(* IEC 61131-3 sources: lasal-git-demo/CPU/LasalDemoProject/Class/TO161, 1 file *)

(* ---- TO161.st ---- *)
#define DEVICE_ID_TO161 1004

#define TO161_ADDR_CYC_WRITE  0
#define TO161_ADDR_CYC_READ   2

#define TO161_WRITE_LENGTH    2
#define TO161_READ_LENGTH     2

(*!
<Class
	Name               = "TO161"
	Revision           = "1.34"
	RealtimeTask       = "false"
	CyclicTask         = "false"
	BackgroundTask     = "false"
	Sigmatek           = "true"
	OSInterface        = "false"
	HighPriority       = "false"
	Automatic          = "false"
	UpdateMode         = "Prescan"
	IconPath           = ".\Class\s-dias.ico"
	SharedCommandTable = "true"
	Objectsize         = "(494,120)"
	Comment            = "This hardware class is used to control the TO161 hardware module with 16 digital outputs.">
	<Channels>
		<Server Name="Output1" Visualized="true" Initialize="false" WriteProtected="false" Retentive="false" Comment="Digital Output 1"/>
		<Server Name="Output10" Visualized="true" Initialize="false" WriteProtected="false" Retentive="false" Comment="Digital Output 10"/>
		<Server Name="Output11" Visualized="true" Initialize="false" WriteProtected="false" Retentive="false" Comment="Digital Output 11"/>
		<Server Name="Output12" Visualized="true" Initialize="false" WriteProtected="false" Retentive="false" Comment="Digital Output 12"/>
		<Server Name="Output13" Visualized="true" Initialize="false" WriteProtected="false" Retentive="false" Comment="Digital Output 13"/>
		<Server Name="Output14" Visualized="true" Initialize="false" WriteProtected="false" Retentive="false" Comment="Digital Output 14"/>
		<Server Name="Output15" Visualized="true" Initialize="false" WriteProtected="false" Retentive="false" Comment="Digital Output 15"/>
		<Server Name="Output16" Visualized="true" Initialize="false" WriteProtected="false" Retentive="false" Comment="Digital Output 16"/>
		<Server Name="Output2" Visualized="true" Initialize="false" WriteProtected="false" Retentive="false" Comment="Digital Output 2"/>
		<Server Name="Output3" Visualized="true" Initialize="false" WriteProtected="false" Retentive="false" Comment="Digital Output 3"/>
		<Server Name="Output4" Visualized="true" Initialize="false" WriteProtected="false" Retentive="false" Comment="Digital Output 4"/>
		<Server Name="Output5" Visualized="true" Initialize="false" WriteProtected="false" Retentive="false" Comment="Digital Output 5"/>
		<Server Name="Output6" Visualized="true" Initialize="false" WriteProtected="false" Retentive="false" Comment="Digital Output 6"/>
		<Server Name="Output7" Visualized="true" Initialize="false" WriteProtected="false" Retentive="false" Comment="Digital Output 7"/>
		<Server Name="Output8" Visualized="true" Initialize="false" WriteProtected="false" Retentive="false" Comment="Digital Output 8"/>
		<Server Name="Output9" Visualized="true" Initialize="false" WriteProtected="false" Retentive="false" Comment="Digital Output 9"/>
		<Server Name="OutputWord" Visualized="true" Initialize="false" WriteProtected="false" Retentive="false" Comment="The digital outputs are displayed in this server in a 16-bit field"/>
		<Server Name="VoltageOkBank1" Visualized="true" Initialize="false" WriteProtected="true" Retentive="false" Comment="Supply voltage ok&#13;&#10;+24V1 (Digital Out 1-8)"/>
		<Server Name="VoltageOkBank2" Visualized="true" Initialize="false" WriteProtected="true" Retentive="false" Comment="Supply voltage ok&#13;&#10;+24V2 (Digital Out 9-16)"/>
	</Channels>
	<RevDoku>
		<Owner Company="Sigmatek" Author="BeiWol"/>
		<Dokumentation Revision="1.34" Date="12.08.2019" Author="LazJos" Company="Sigmatek" Description="Added support for HWAlarms."/>
		<Dokumentation Revision="1.33" Date="09.01.2019" Author="FurDom" Company="Sigmatek" Description="Added function for Spi Write in SdiasBase class."/>
		<Dokumentation Revision="1.32" Date="08.06.2018" Author="RamAnd" Company="Sigmatek" Description="LASAL Hardware Description (.lhd) file has been updated."/>
		<Dokumentation Revision="1.31" Date="16.05.2017" Author="RamAnd" Company="Sigmatek" Description="When adding an SDO (i.e. via ReadSPIData) from background priority it was possible that the adding process got interrupted by receiving the answer to this SDO which is handled in cyclic priority. In the error case the answer was unexpected and therefore ignored. Then the class signals a timeout while waiting for the answer, which already arrived before waiting for it. Added mutex and changed instruction order to prevent this error."/>
		<Dokumentation Revision="1.30" Date="12.07.2016" Author="SeiChr" Company="Sigmatek" Description="Added Values for the total Current calculation. SA 31571"/>
		<Dokumentation Revision="1.29" Date="01.03.2016" Author="EisMic" Company="Sigmatek" Description="Corrected BoundExceed Error in base class at Write method of LEDControl Server when Place = LSL_DEACTIVATED."/>
		<Dokumentation Revision="1.28" Date="22.06.2015" Author="EisMic" Company="Sigmatek" Description="The servers FPGAVersion, SerialNo, Device ID and status and input servers are now not reset anymore when the module is disconnected.&#13;&#10;Outputs are now written to the hardware in any case after a reconnect."/>
		<Dokumentation Revision="1.27" Date="27.05.2015" Author="EisMic" Company="Sigmatek" Description="Corrected ConnectEvent Method that outputs are set after reconnect."/>
		<Dokumentation Revision="1.26" Date="16.04.2015" Author="EisMic&#13;&#10;LanSte" Company="Sigmatek" Description="Added support for visualisation in graphical hardware editor.&#13;&#10;Added support for calculating resources for graphical hardware editor."/>
		<Dokumentation Revision="1.25" Date="17.03.2015" Author="RamAnd" Company="Sigmatek" Description="Added HW Version for sdias clients."/>
		<Dokumentation Revision="1.24" Date="11.02.2015" Author="PieSte" Company="Sigmatek" Description="Corrected read spi data for hardwaretree in methode GetSPIDataFromID from baseclass."/>
		<Dokumentation Revision="1.23" Date="03.12.2014" Author="PieSte" Company="Sigmatek" Description="Add OutputByte in .lhd file."/>
		<Dokumentation Revision="1.22" Date="18.11.2014" Author="PieSte" Company="Sigmatek" Description="Added possibility  to read more data from spi flash then one sdo access.&#13;&#10;Set methode GetDeviceID to global.&#13;&#10;Add methode to calculate checksum of spi flash."/>
		<Dokumentation Revision="1.21" Date="09.07.2014" Author="EisMic" Company="Sigmatek" Description="Added support for reading hardware diagnosis and hardwaretree entry."/>
		<Dokumentation Revision="1.20" Date="20.01.2014" Author="PieSte" Company="Sigmatek" Description="Read Client Required and Place in Init SdiasBase"/>
		<Dokumentation Revision="1.10" Date="05.12.2013" Author="RamAnd" Company="Sigmatek" Description="Changed login mechanism to sdias manager class to be independent of bus accesses."/>
		<Dokumentation Revision="1.0" Date="25.07.2013" Author="BeiWol" Company="Sigmatek" Description="First library version"/>
	</RevDoku>
	<Network Name="TO161">
		<!-- List of Components in this network -->
		<Components>
			<Object
				Name       = "_base"
				Class      = "SdiasBase"
				Position   = "(218,120)"
				Visualized = "true">
				<Channels>
					<Server Name="ClassState"/>
					<Server Name="DeviceID"/>
					<Server Name="FPGAVersion"/>
					<Server Name="HwVersion"/>
					<Server Name="LEDControl" Value="0"/>
					<Server Name="RetryCounter"/>
					<Server Name="SDOState"/>
					<Server Name="SerialNo"/>
					<Client Name="Place" Value="0"/>
					<Client Name="Required" Value="1"/>
					<Client Name="SdiasIn"/>
					<Client Name="ToStdLib"/>
				</Channels>
			</Object>
		</Components>
		<Comments>
		</Comments>
		<!-- List of Connections in this network -->
		<Connections>
			<Connection Source="this.ClassState" Destination="_base.ClassState" Vertices="(804,210),(632,210),"/>
			<Connection Source="this.DeviceID" Destination="_base.DeviceID" Vertices="(804,270),(632,270),"/>
			<Connection Source="this.SerialNo" Destination="_base.SerialNo" Vertices="(804,450),(632,450),"/>
			<Connection Source="this.RetryCounter" Destination="_base.RetryCounter" Vertices="(804,510),(632,510),"/>
			<Connection Source="_base.SdiasIn" Destination="this.SdiasIn" Vertices="(218,210),(38,210),"/>
			<Connection Source="_base.Place" Destination="this.Place" Vertices="(218,270),(38,270),"/>
			<Connection Source="_base.Required" Destination="this.Required" Vertices="(218,330),(38,330),"/>
			<Connection Source="this.LEDControl" Destination="_base.LEDControl" Vertices="(804,570),(632,570),"/>
			<Connection Source="this.FPGAVersion" Destination="_base.FPGAVersion" Vertices="(804,330),(632,330),"/>
			<Connection Source="this.HwVersion" Destination="_base.HwVersion" Vertices="(804,390),(632,390),"/>
		</Connections>
		<!-- Headerfiles -->
		<Options>
		</Options>
	</Network>
</Class>
*)
#pragma using SdiasBase

TO161 : CLASS
: SdiasBase
	TYPE
	  t_VoltageOk : BINT
	  [
	    1 Ok24V1,
	    2 Ok24V2,
	  ];
	END_TYPE
  //Servers:
	Output1 	: SvrCh_DINT;
	Output2 	: SvrCh_DINT;
	Output3 	: SvrCh_DINT;
	Output4 	: SvrCh_DINT;
	Output5 	: SvrCh_DINT;
	Output6 	: SvrCh_DINT;
	Output7 	: SvrCh_DINT;
	Output8 	: SvrCh_DINT;
	Output9 	: SvrCh_DINT;
	Output10 	: SvrCh_DINT;
	Output11 	: SvrCh_DINT;
	Output12 	: SvrCh_DINT;
	Output13 	: SvrCh_DINT;
	Output14 	: SvrCh_DINT;
	Output15 	: SvrCh_DINT;
	Output16 	: SvrCh_DINT;
	OutputWord 	: SvrCh_BDINT;
	VoltageOkBank1 	: SvrCh_DINT;
	VoltageOkBank2 	: SvrCh_DINT;
  //Clients:
  //Variables:
		bdOutputBitsOld : BDINT
		[
		];
			//! <Variable Comment="Merker for old OutputStatus." Name="bdOutputBitsOld"/>
		pReadData 	: ^UINT;			//! <Variable Comment="Read-Data from the Module." Name="pReadData"/>
		pWriteData 	: ^UINT;			//! <Variable Comment="WriteData of the Module." Name="pWriteData"/>
  //Functions:
				//! <Function Comment="Realtime Update Methode which runs in PreScan." Name="UpdateRt"/>
	FUNCTION VIRTUAL GLOBAL UpdateRt;
				//! <Function Comment="Realtime Update Methode which runs in PostScan." Name="UpdateRtPostScan"/>
	FUNCTION VIRTUAL GLOBAL UpdateRtPostScan;
				//! <Function Comment="Methode is called if this Module gets connected." Name="ConnectEvent"/>
	FUNCTION VIRTUAL GLOBAL ConnectEvent;
				//! <Function Comment="Methode is called if this Module gets disconnected." Name="DisconnectEvent"/>
	FUNCTION VIRTUAL GLOBAL DisconnectEvent;
				//! <Function Comment="This Methode should is used, to check the DeviceID of the Module." Name="CheckDeviceID"/>
	FUNCTION VIRTUAL GLOBAL CheckDeviceID
		VAR_INPUT
			udID2Check 	: UDINT;			//! <Variable Comment="Device ID of connected Module." Name="CheckDeviceID.udID2Check"/>
		END_VAR
		VAR_OUTPUT
			bIsOK 	: BOOL;			//! <Variable Comment="FALSE = Wrong DeviceID for Module&#13;&#10;TRUE  = DeviceID of Module is correct" Name="CheckDeviceID.bIsOK"/>
		END_VAR;

	FUNCTION VIRTUAL GetTaskCfg
		VAR_OUTPUT
			TaskCfg 	: BDINT;			//! <Variable Comment="Select which tasks will be available for this module:&#13;&#10;Bit0..Realtime PreScan&#13;&#10;Bit1..Realtime PostScan&#13;&#10;Bit2..Cyclic&#13;&#10;&#13;&#10;e.g. if only realtime postscan is needed:&#13;&#10;2#010" Name="GetTaskCfg.TaskCfg"/>
		END_VAR;

	FUNCTION VIRTUAL GetDeviceID
		VAR_OUTPUT
			output 	: UDINT;
		END_VAR;

	FUNCTION VIRTUAL GLOBAL Output1::Write
		VAR_INPUT
			input (EAX) 	: DINT;
		END_VAR
		VAR_OUTPUT
			result (EAX) 	: DINT;
		END_VAR;

	FUNCTION VIRTUAL GLOBAL Output2::Write
		VAR_INPUT
			input (EAX) 	: DINT;
		END_VAR
		VAR_OUTPUT
			result (EAX) 	: DINT;
		END_VAR;

	FUNCTION VIRTUAL GLOBAL Output3::Write
		VAR_INPUT
			input (EAX) 	: DINT;
		END_VAR
		VAR_OUTPUT
			result (EAX) 	: DINT;
		END_VAR;

	FUNCTION VIRTUAL GLOBAL Output4::Write
		VAR_INPUT
			input (EAX) 	: DINT;
		END_VAR
		VAR_OUTPUT
			result (EAX) 	: DINT;
		END_VAR;

	FUNCTION VIRTUAL GLOBAL Output5::Write
		VAR_INPUT
			input (EAX) 	: DINT;
		END_VAR
		VAR_OUTPUT
			result (EAX) 	: DINT;
		END_VAR;

	FUNCTION VIRTUAL GLOBAL Output6::Write
		VAR_INPUT
			input (EAX) 	: DINT;
		END_VAR
		VAR_OUTPUT
			result (EAX) 	: DINT;
		END_VAR;

	FUNCTION VIRTUAL GLOBAL Output7::Write
		VAR_INPUT
			input (EAX) 	: DINT;
		END_VAR
		VAR_OUTPUT
			result (EAX) 	: DINT;
		END_VAR;

	FUNCTION VIRTUAL GLOBAL Output8::Write
		VAR_INPUT
			input (EAX) 	: DINT;
		END_VAR
		VAR_OUTPUT
			result (EAX) 	: DINT;
		END_VAR;

	FUNCTION VIRTUAL GLOBAL Output9::Write
		VAR_INPUT
			input (EAX) 	: DINT;
		END_VAR
		VAR_OUTPUT
			result (EAX) 	: DINT;
		END_VAR;

	FUNCTION VIRTUAL GLOBAL Output10::Write
		VAR_INPUT
			input (EAX) 	: DINT;
		END_VAR
		VAR_OUTPUT
			result (EAX) 	: DINT;
		END_VAR;

	FUNCTION VIRTUAL GLOBAL Output11::Write
		VAR_INPUT
			input (EAX) 	: DINT;
		END_VAR
		VAR_OUTPUT
			result (EAX) 	: DINT;
		END_VAR;

	FUNCTION VIRTUAL GLOBAL Output12::Write
		VAR_INPUT
			input (EAX) 	: DINT;
		END_VAR
		VAR_OUTPUT
			result (EAX) 	: DINT;
		END_VAR;

	FUNCTION VIRTUAL GLOBAL Output13::Write
		VAR_INPUT
			input (EAX) 	: DINT;
		END_VAR
		VAR_OUTPUT
			result (EAX) 	: DINT;
		END_VAR;

	FUNCTION VIRTUAL GLOBAL Output14::Write
		VAR_INPUT
			input (EAX) 	: DINT;
		END_VAR
		VAR_OUTPUT
			result (EAX) 	: DINT;
		END_VAR;

	FUNCTION VIRTUAL GLOBAL Output15::Write
		VAR_INPUT
			input (EAX) 	: DINT;
		END_VAR
		VAR_OUTPUT
			result (EAX) 	: DINT;
		END_VAR;

	FUNCTION VIRTUAL GLOBAL Output16::Write
		VAR_INPUT
			input (EAX) 	: DINT;
		END_VAR
		VAR_OUTPUT
			result (EAX) 	: DINT;
		END_VAR;

	FUNCTION VIRTUAL GLOBAL OutputWord::Write
		VAR_INPUT
			input (EAX) 	: BDINT;
		END_VAR
		VAR_OUTPUT
			result (EAX) 	: BDINT;
		END_VAR;
  //Tables:
	FUNCTION @STD
		VAR_OUTPUT
			ret_code	: CONFSTATES;
		END_VAR;
	FUNCTION GLOBAL TAB @CT_;
END_CLASS;

FUNCTION VIRTUAL GLOBAL TO161::UpdateRt
  VAR
    VoltageOkTmp  : t_VoltageOk;
  END_VAR

  VoltageOkTmp := (pReadData^)$BINT;

  VoltageOkBank1 := VoltageOkTmp.Ok24V1;
  VoltageOkBank2 := VoltageOkTmp.Ok24V2;

END_FUNCTION

FUNCTION VIRTUAL GLOBAL TO161::UpdateRtPostScan

  if OutputWord <> bdOutputBitsOld then
    pWriteData^ := OutputWord$BINT;

    bdOutputBitsOld := OutputWord;
  end_if;

END_FUNCTION

FUNCTION VIRTUAL GLOBAL TO161::CheckDeviceID
	VAR_INPUT
		udID2Check 	: UDINT;
	END_VAR
	VAR_OUTPUT
		bIsOK 	: BOOL;
	END_VAR

  //look if it is right hardware
	if ( udID2Check <> DEVICE_ID_TO161 ) then
		bIsOK := FALSE;
	else
    bIsOK := TRUE;
	end_if;

END_FUNCTION

FUNCTION VIRTUAL GLOBAL TO161::ConnectEvent

  // start the accesses on the SDIAS (initialize the control byte in the DPRAM)
  if DefaultAccesses.ReadAccess.pControlByte then
    pReadData := DefaultAccesses.ReadAccess.pData$^UINT;

    DefaultAccesses.ReadAccess.pControlByte^.EnableDO := TRUE;
  else
    eInitState := _DOHandleInvalid;
    return;
  end_if;

  if DefaultAccesses.WriteAccess.pControlByte then
    pWriteData := DefaultAccesses.WriteAccess.pData$^UINT;

    DefaultAccesses.WriteAccess.pControlByte^.EnableDO := TRUE;
  else
    eInitState := _DOHandleInvalid;
    return;
  end_if;

  //Set to write outputs at first access and after reconnect
  bdOutputBitsOld := NOT OutputWord;

  // module is ok
  eInitState := _ClassOk;

END_FUNCTION

FUNCTION VIRTUAL GLOBAL TO161::DisconnectEvent

  //Reset Write-Memory
  if pWriteData then
    _memset(dest := pWriteData, usByte := 0, cntr := sizeof(pWriteData^));
  end_if;

  // reset general module information shown on servers
  SdiasBase::DisconnectEvent();

  VoltageOkBank1 := 0;
  VoltageOkBank2 := 0;

END_FUNCTION

FUNCTION VIRTUAL GLOBAL TO161::Output1::Write
	VAR_INPUT
		input (EAX) 	: DINT;
	END_VAR
	VAR_OUTPUT
		result (EAX) 	: DINT;
	END_VAR

  if input then
    result  := 1;
    Output1 := 1;
    OutputWord.1  := 1;
  else
    result  := 0;
    Output1 := 0;
    OutputWord.1  := 0;
  end_if;

END_FUNCTION

FUNCTION VIRTUAL GLOBAL TO161::Output2::Write
	VAR_INPUT
		input (EAX) 	: DINT;
	END_VAR
	VAR_OUTPUT
		result (EAX) 	: DINT;
	END_VAR

  if input then
    result  := 1;
    Output2 := 1;
    OutputWord.2  := 1;
  else
    result  := 0;
    Output2 := 0;
    OutputWord.2  := 0;
  end_if;

END_FUNCTION

FUNCTION VIRTUAL GLOBAL TO161::Output3::Write
	VAR_INPUT
		input (EAX) 	: DINT;
	END_VAR
	VAR_OUTPUT
		result (EAX) 	: DINT;
	END_VAR

  if input then
    result  := 1;
    Output3 := 1;
    OutputWord.3  := 1;
  else
    result  := 0;
    Output3 := 0;
    OutputWord.3  := 0;
  end_if;

END_FUNCTION

FUNCTION VIRTUAL GLOBAL TO161::Output4::Write
	VAR_INPUT
		input (EAX) 	: DINT;
	END_VAR
	VAR_OUTPUT
		result (EAX) 	: DINT;
	END_VAR

  if input then
    result  := 1;
    Output4 := 1;
    OutputWord.4  := 1;
  else
    result  := 0;
    Output4 := 0;
    OutputWord.4  := 0;
  end_if;

END_FUNCTION

FUNCTION VIRTUAL GLOBAL TO161::Output5::Write
	VAR_INPUT
		input (EAX) 	: DINT;
	END_VAR
	VAR_OUTPUT
		result (EAX) 	: DINT;
	END_VAR

  if input then
    result  := 1;
    Output5 := 1;
    OutputWord.5  := 1;
  else
    result  := 0;
    Output5 := 0;
    OutputWord.5  := 0;
  end_if;

END_FUNCTION

FUNCTION VIRTUAL GLOBAL TO161::Output6::Write
	VAR_INPUT
		input (EAX) 	: DINT;
	END_VAR
	VAR_OUTPUT
		result (EAX) 	: DINT;
	END_VAR

  if input then
    result  := 1;
    Output6 := 1;
    OutputWord.6  := 1;
  else
    result  := 0;
    Output6 := 0;
    OutputWord.6  := 0;
  end_if;

END_FUNCTION

FUNCTION VIRTUAL GLOBAL TO161::Output7::Write
	VAR_INPUT
		input (EAX) 	: DINT;
	END_VAR
	VAR_OUTPUT
		result (EAX) 	: DINT;
	END_VAR

  if input then
    result  := 1;
    Output7 := 1;
    OutputWord.7  := 1;
  else
    result  := 0;
    Output7 := 0;
    OutputWord.7  := 0;
  end_if;

END_FUNCTION

FUNCTION VIRTUAL GLOBAL TO161::Output8::Write
	VAR_INPUT
		input (EAX) 	: DINT;
	END_VAR
	VAR_OUTPUT
		result (EAX) 	: DINT;
	END_VAR

  if input then
    result  := 1;
    Output8 := 1;
    OutputWord.8  := 1;
  else
    result  := 0;
    Output8 := 0;
    OutputWord.8  := 0;
  end_if;

END_FUNCTION

FUNCTION VIRTUAL GLOBAL TO161::Output9::Write
	VAR_INPUT
		input (EAX) 	: DINT;
	END_VAR
	VAR_OUTPUT
		result (EAX) 	: DINT;
	END_VAR

  if input then
    result  := 1;
    Output9 := 1;
    OutputWord.9  := 1;
  else
    result  := 0;
    Output9 := 0;
    OutputWord.9  := 0;
  end_if;

END_FUNCTION

FUNCTION VIRTUAL GLOBAL TO161::Output10::Write
	VAR_INPUT
		input (EAX) 	: DINT;
	END_VAR
	VAR_OUTPUT
		result (EAX) 	: DINT;
	END_VAR

  if input then
    result  := 1;
    Output10 := 1;
    OutputWord.10  := 1;
  else
    result  := 0;
    Output10 := 0;
    OutputWord.10  := 0;
  end_if;

END_FUNCTION

FUNCTION VIRTUAL GLOBAL TO161::Output11::Write
	VAR_INPUT
		input (EAX) 	: DINT;
	END_VAR
	VAR_OUTPUT
		result (EAX) 	: DINT;
	END_VAR

  if input then
    result  := 1;
    Output11 := 1;
    OutputWord.11  := 1;
  else
    result  := 0;
    Output11 := 0;
    OutputWord.11  := 0;
  end_if;

END_FUNCTION

FUNCTION VIRTUAL GLOBAL TO161::Output12::Write
	VAR_INPUT
		input (EAX) 	: DINT;
	END_VAR
	VAR_OUTPUT
		result (EAX) 	: DINT;
	END_VAR

  if input then
    result  := 1;
    Output12 := 1;
    OutputWord.12  := 1;
  else
    result  := 0;
    Output12 := 0;
    OutputWord.12  := 0;
  end_if;

END_FUNCTION

FUNCTION VIRTUAL GLOBAL TO161::Output13::Write
	VAR_INPUT
		input (EAX) 	: DINT;
	END_VAR
	VAR_OUTPUT
		result (EAX) 	: DINT;
	END_VAR

  if input then
    result  := 1;
    Output13 := 1;
    OutputWord.13  := 1;
  else
    result  := 0;
    Output13 := 0;
    OutputWord.13  := 0;
  end_if;

END_FUNCTION

FUNCTION VIRTUAL GLOBAL TO161::Output14::Write
	VAR_INPUT
		input (EAX) 	: DINT;
	END_VAR
	VAR_OUTPUT
		result (EAX) 	: DINT;
	END_VAR

  if input then
    result  := 1;
    Output14 := 1;
    OutputWord.14  := 1;
  else
    result  := 0;
    Output14 := 0;
    OutputWord.14  := 0;
  end_if;

END_FUNCTION

FUNCTION VIRTUAL GLOBAL TO161::Output15::Write
	VAR_INPUT
		input (EAX) 	: DINT;
	END_VAR
	VAR_OUTPUT
		result (EAX) 	: DINT;
	END_VAR

  if input then
    result  := 1;
    Output15 := 1;
    OutputWord.15  := 1;
  else
    result  := 0;
    Output15 := 0;
    OutputWord.15  := 0;
  end_if;

END_FUNCTION

FUNCTION VIRTUAL GLOBAL TO161::Output16::Write
	VAR_INPUT
		input (EAX) 	: DINT;
	END_VAR
	VAR_OUTPUT
		result (EAX) 	: DINT;
	END_VAR

  if input then
    result  := 1;
    Output16 := 1;
    OutputWord.16  := 1;
  else
    result  := 0;
    Output16 := 0;
    OutputWord.16  := 0;
  end_if;

END_FUNCTION

FUNCTION VIRTUAL GLOBAL TO161::OutputWord::Write
	VAR_INPUT
		input (EAX) 	: BDINT;
	END_VAR
	VAR_OUTPUT
		result (EAX) 	: BDINT;
	END_VAR

  if( input$hint <> OutputWord$hint)then
    Output1 :=  (input and 2#1)$DINT;
    Output2 :=  (input and 2#10)$DINT shr 1;
    Output3 :=  (input and 2#100)$DINT shr 2;
    Output4 :=  (input and 2#1000)$DINT shr 3;
    Output5 :=  (input and 2#10000)$DINT shr 4;
    Output6 :=  (input and 2#100000)$DINT shr 5;
    Output7 :=  (input and 2#1000000)$DINT shr 6;
    Output8 :=  (input and 2#10000000)$DINT shr 7;
    Output9 :=  (input and 2#100000000)$DINT shr 8;
    Output10 := (input and 2#1000000000)$DINT shr 9;
    Output11 := (input and 2#10000000000)$DINT shr 10;
    Output12 := (input and 2#100000000000)$DINT shr 11;
    Output13 := (input and 2#1000000000000)$DINT shr 12;
    Output14 := (input and 2#10000000000000)$DINT shr 13;
    Output15 := (input and 2#100000000000000)$DINT shr 14;
    Output16 := (input and 2#1000000000000000)$DINT shr 15;
  end_if;
 	OutputWord := result := input;

END_FUNCTION

FUNCTION VIRTUAL TO161::GetTaskCfg
	VAR_OUTPUT
		TaskCfg 	: BDINT;
	END_VAR

  TaskCfg := SDIAS_TASK_MASK_RT_PRE OR SDIAS_TASK_MASK_RT_POST;

END_FUNCTION

FUNCTION VIRTUAL TO161::GetDeviceID
	VAR_OUTPUT
		output 	: UDINT;
	END_VAR

  output := DEVICE_ID_TO161;

END_FUNCTION
